(* PLC project UML_SC_CoffeeMachine.project, CODESYS CODESYS V3.5 SP18 Patch 4 *)
(* stored: creationDateTime 2023-10-22T20:37:55.9701005, modificationDateTime 2021-04-08T20:07:10 *)

{attribute 'no-analysis'}
{attribute 'reduced_bp_set'}
PROGRAM Kaffemaschine
  VAR
    bMakeCoffee : BOOL := FALSE;
    bShutDown : BOOL := FALSE;
    bPowerUp : BOOL := FALSE;
    nGrind : INT := 0;
    nHeat : INT := 20;
    nFoam : INT := 0;
    {attribute 'implicit_state_chart_struct'}
    UML_SC_Kaffemaschine : _UML_SC_7cc42eb0dc6d4e02ab5b1296bec80ed6;
    {attribute 'implicit_state_chart_struct'}
    UML_SC_ActHeat : _UML_SC_9e3c3d30f6c84991be9f932f948dff00;
  END_VAR

            
          

ACTION ActEntry:
                
              
END_ACTION

ACTION ActShutdown:
                bShutDown := FALSE;
bPowerUp := FALSE;
              
END_ACTION

ACTION CoffeeReady:
                bMakeCoffee := FALSE;
nGrind := 0;
nHeat := 20;
nFoam := 0;
              
END_ACTION

ACTION ActDo:
                nGrind := nGrind + 10;
              
END_ACTION

ACTION ActHeat:
                
              
END_ACTION

ACTION ActFoam:
                nFoam := nFoam + 5;
              
END_ACTION
END_PROGRAM
